Yaskawa INFORM job: TEST-WELD-STATION-2.JBI

/JOB
//NAME TEST-WELD-STATION-2
//POS
///NPOS 5,5,5,2,0,5
///TOOL 0
///POSTYPE PULSE
///PULSE
C00000=90902,7535,9485,-58400,43717,82890
C00001=90902,7535,9485,-58400,43717,82890
C00002=91129,-5534,-21902,-89083,49459,101717
C00003=91652,-5566,-22271,-89546,49769,101989
C00004=91033,-5293,-22071,-89378,49363,101938
BC00000=208121
BC00001=208121
BC00002=208121
BC00003=208120
BC00004=208120
EC00000=-6
EC00001=246513
EC00002=-2604
EC00003=0
EC00004=0
///POSTYPE BASE
///RECTAN
///RCONF 1,0,0,0,1,0,0,0,0,0,0,0,0,0,0,0,0,0,0,0,0,0,0,0
P00125=1436.096,1808.596,415.287,-4.2393,5.8699,103.4291
P00126=1375.000,1808.603,361.298,-4.2419,5.8697,103.4275
///POSTYPE ANGLE
///ANGLE
EX00000=0.0000
EX00045=-90.0000
EX00046=-180.0000
EX00047=-270.0000
EX00048=-365.0000
//INST
///DATE 2018/10/30 16:25
///ATTR SC,RW
///GROUP1 RB1,BS1
///GROUP2 ST2
NOP
MOVJ C00000 BC00000 VJ=10.00  +MOVJ EC00000 VJ=100.00
MOVJ C00001 BC00001 VJ=10.00  +MOVJ EC00001 VJ=100.00
SMOVL C00002 BC00002 V=83.3  +MOVJ EC00002
SMOVL P126 V=83.3 PL=0  +MOVJ EX000
SREFP 1 C00003 BC00003  +REFP EC00003
SREFP 2 C00004 BC00004  +REFP EC00004
DOUT OT#(656) ON
MACRO1 MJ#(5) ARGF5
ARCON ASF#(1)
SACORON TF TCH#(3) TV=I001
SMOVC P126 V=83.3 PL=0  +MOVJ EX000
SMOVC P126 V=I000  +MOVJ EX045
SMOVC P126 V=I000  +MOVJ EX046
SMOVC P126 V=I000  +MOVJ EX047
SMOVC P126 V=I000  +MOVJ EX048
SWVOF
SACOROF
ARCOF
MACRO1 MJ#(5) ARGF5
TIMER T=6.00
DOUT OT#(656) OFF
SMOVL P125 V=83.3 PL=0  +MOVJ EX048
END
